INTERFACE INTERNAL I_ExecuteNode EXTENDS I_Debug;

METHOD INTERNAL Attach : Result
VAR_INPUT
	iExecute		: I_ExecuteNode;
END_VAR
END_METHOD

METHOD INTERNAL Exe
VAR_INPUT
END_VAR
END_METHOD

PROPERTY INTERNAL State : Result
GET
END_GET
SET
END_SET
END_PROPERTY

END_INTERFACE

(* stored: Version 1.1.0.1
   Itf I_ExecuteNode: Id {8b79cbd5-d7c4-4c85-85bb-38aa830221fc}
   Method Attach: Id {579bbb33-36fc-4df5-b518-286df0af34fa}
   Method Exe: Id {8d48a61b-dcd6-4e45-8916-d669dffef6c5}
   Property State: Id {275348de-dbc3-4cde-8a89-26f662986a85}
   Get Get: Id {35fdd807-57a9-4770-a7d0-768abbb81aa9}
   Set Set: Id {27c80dc8-963d-4f70-96df-3dd9dddd17a4} *)
